
FUNCTION CB_int_to_sint : INT

TITLE = ' Convert an integer into a word '
VERSION : '1.0'
AUTHOR  : CB
NAME    : intToByt
FAMILY  : TNI

VAR_INPUT
    IN : INT;
END_VAR

BEGIN

CB_int_to_sint := IN;

END_FUNCTION
